TYPE PLCOpenCallInternal :
STRUCT
	_state : PLCOpenCallState;
	_Command: IPLCOpenCommand;
	_abort: BOOL;
	_execute: BOOL;
	_break:BOOL;
	_RemoteStatus: PLCOPENSTATUSBASE;
	_self :IPLCOpenCall;
END_STRUCT
END_TYPE

(* stored: Version 1.1.0.1, ProductVersion 3.1.4024.12
   DUT PLCOpenCallInternal: Id {a493e5a4-f6ba-450d-b862-4481c25cddf0} *)
